{attribute 'GeneratedUsingTerminal: EK1122-0000-0018'}
{attribute addProperty BoxType "EK1122-0000-0018"}
{attribute addProperty Id "Beckhoff_EP4xxxsub_EK1100EK1100_AB5A94672A_0001_EP4174_0002_0016EP4174_F6F08E1219A_0002_EP4174_0002_0017EP4174_F6F08E1219A_0003_EP4174_0002_0018EP4174_F6F08E1219A_0004_EP4174_0002_0019EP4174_F6F08E1219A_0005_EP4314_1002_0016EP4314_F6FCB00838A_0006_EP4374_0002_0016EP4374_002067C436A_0007_EP4374_0002_0017EP4374_8019271A36A_0008_EP4374_0002_0018EP4374_8019271A36A_0009_EP4374_0002_0019EP4374_8019271A36A_0010_EP4378_1022_0017EP4378_D09B5E9776"}
{attribute addProperty CRC "4193978453"}
{attribute addProperty Size "336"}
TYPE Beckhoff_EP4xxxEK1122_F9FB0855 EXTENDS EK1122_AB5A9467 :
STRUCT
	{attribute addProperty Name "Beckhoff_EP4xxxsub_EK1100"}
	Beckhoff_EP4xxxsub_EK1100 : EK1100_AB5A9467;
	{attribute addProperty Name "A_0001_EP4174_0002_0016"}
	A_0001_EP4174_0002_0016 : EP4174_F6F08E12;
	{attribute addProperty Name "A_0002_EP4174_0002_0017"}
	A_0002_EP4174_0002_0017 : EP4174_F6F08E12;
	{attribute addProperty Name "A_0003_EP4174_0002_0018"}
	A_0003_EP4174_0002_0018 : EP4174_F6F08E12;
	{attribute addProperty Name "A_0004_EP4174_0002_0019"}
	A_0004_EP4174_0002_0019 : EP4174_F6F08E12;
	{attribute addProperty Name "A_0005_EP4314_1002_0016"}
	A_0005_EP4314_1002_0016 : EP4314_F6FCB008;
	{attribute addProperty Name "A_0006_EP4374_0002_0016"}
	A_0006_EP4374_0002_0016 : EP4374_002067C4;
	{attribute addProperty Name "A_0007_EP4374_0002_0017"}
	A_0007_EP4374_0002_0017 : EP4374_8019271A;
	{attribute addProperty Name "A_0008_EP4374_0002_0018"}
	A_0008_EP4374_0002_0018 : EP4374_8019271A;
	{attribute addProperty Name "A_0009_EP4374_0002_0019"}
	A_0009_EP4374_0002_0019 : EP4374_8019271A;
	{attribute addProperty Name "A_0010_EP4378_1022_0017"}
	A_0010_EP4378_1022_0017 : EP4378_D09B5E97;
END_STRUCT
END_TYPE

(* stored: Version 1.2.0.0, ProductVersion 3.1.4024.9
   DUT Beckhoff_EP4xxxEK1122_F9FB0855: Id {36c04a66-18c6-4c1c-8291-3c7345d298c8} *)
